PROGRAM P_Demo_FB_DMXDiscUnMute
VAR
    fbDiscUnMute      : FB_DMXDiscUnMute;             // 复位设备 mute 标志
    stDmxCmdBuffer    : ST_DMXCommandBuffer;          // 与通讯 FB 共用
    wTargetManufId    : WORD := 16#4241;              // 目标灯具厂商 ID
    dwTargetDeviceId  : DWORD := 16#12131415;         // 目标灯具设备 ID
    byTargetPort      : BYTE := 0;                    // 根设备通道 0
    bDoUnMute         : BOOL := FALSE;                // 在线给一次上升沿触发
    bBusy             : BOOL;
    bError            : BOOL;
    udiErrId          : UDINT;
    wCtrlField        : WORD;                         // 设备返回的控制字段
END_VAR

// ============================================================
// Tc2_DMX.FB_DMXDiscUnMute 演示程序
// ============================================================
// 场景：自定义发现流程结束后，把先前 mute 掉的设备全部恢复，以便下一轮搜索或让其它控制器也能发现。
// 价值：把 RDM 发现协议中的 un-mute 步骤暴露为单独 FB，配合 Mute / UniqueBranch 实现完全自定义的发现策略。
// 验证：先用 FB_DMXDiscMute 把目标设备 mute，再给 bDoUnMute 一次上升沿 -> bBusy 短暂 TRUE -> 回 FALSE 后对该设备发 UniqueBranch 应又能得到响应。
// 验证步骤：
//   1. 右键 PLC 项目下 POUs 文件夹 → Add → Existing Item → 选本 .TcPOU 文件
//   2. 引用 Tc2_DMX；同项目里放一个 FB_EL6851CommunicationEx 实例并共用 stDmxCmdBuffer（非 CycleMode）
//   3. 编译 → 登录 → 运行；按上方『验证』行在线给上升沿观察
// ============================================================

fbDiscUnMute(
    bStart                     := bDoUnMute,
    wDestinationManufacturerId := wTargetManufId,
    dwDestinationDeviceId      := dwTargetDeviceId,
    byPortId                   := byTargetPort,
    dwOptions                  := 0,
    stCommandBuffer            := stDmxCmdBuffer,
    bBusy                      => bBusy,
    bError                     => bError,
    udiErrorId                 => udiErrId,
    wControlField              => wCtrlField
);

END_PROGRAM

(* stored: Version 1.1.0.1, ProductVersion 3.1.4024.5
   POU P_Demo_FB_DMXDiscUnMute: Id {1ef1986a-0c8b-59aa-a163-79f57036f590}, SpecialFunc None *)
